
FUNCTION CB_mul_t_sint : TIME


TITLE = ' Multiplying a time '
VERSION : '1.0'
AUTHOR  : CB
NAME    : mulTiSin
FAMILY  : TNI

VAR_INPUT
    IN0 : TIME;
    IN1 : INT;
END_VAR

BEGIN
    CB_mul_t_sint := IN0 * IN1;
END_FUNCTION
